// TIA Portal project "convergestation_Ronaldo" (V18)

(* hardware
DEVICE "S7-1200 station_1"  S7-1200 Station
   slot 0: "Rack_0"  S7-1200 Rack  Rack  V1.0
   slot 1: "Automacao_convergestation"  CPU 1214C DC/DC/DC  6ES7 214-1AG40-0XB0  V4.4
   slot 2: "DI 8/DQ 8x24VDC_1"  6ES7 223-1BH32-0XB0  V2.0
*)

// ===== PLC "Automacao_convergestation"  CPU 1214C DC/DC/DC =====

VAR_GLOBAL   // PLC tag table "Default tag table"
   "Emergência" AT %I0.0 : Bool;
   "Botão Start" AT %I0.1 : Bool;
   "Botão Stop" AT %I0.2 : Bool;
   "Botão Reset" AT %I0.3 : Bool;
   "Manual" AT %I0.4 : Bool;
   "Automático" AT %I0.5 : Bool;
   "Contador" AT %QD30 : DInt;
   "Clock_Byte" AT %MB0 : Byte;
   "Clock_10Hz" AT %M0.0 : Bool;
   "Clock_5Hz" AT %M0.1 : Bool;
   "Clock_2.5Hz" AT %M0.2 : Bool;
   "Clock_2Hz" AT %M0.3 : Bool;
   "Clock_1.25Hz" AT %M0.4 : Bool;
   "Clock_1Hz" AT %M0.5 : Bool;
   "Clock_0.625Hz" AT %M0.6 : Bool;
   "Clock_0.5Hz" AT %M0.7 : Bool;
   "Sen. Esteira 01" AT %I0.6 : Bool;
   "Sen. Esteira 02" AT %I0.7 : Bool;
   "Sen. Transf. 01" AT %I1.0 : Bool;
   "Sen. Transf. 02" AT %I1.1 : Bool;
   "Sen.  de Saída" AT %I1.2 : Bool;
   "Esteira 01" AT %Q0.0 : Bool;
   "Esteira 02" AT %Q0.1 : Bool;
   "Esteira de Saída" AT %Q0.2 : Bool;
   "Carregar 01" AT %Q0.3 : Bool;
   "Carregar 02" AT %Q0.4 : Bool;
   "Descarregar 01" AT %Q0.5 : Bool;
   "Descarregar 02" AT %Q0.6 : Bool;
   "Transf. 01 Direita" AT %Q0.7 : Bool;
   "Transf. 02 Direita" AT %Q1.0 : Bool;
   "Transf. 01 Esquerda" AT %Q1.1 : Bool;
   "Transf. 02 Esquerda" AT %Q1.2 : Bool;
   "Led Verde" AT %Q1.3 : Bool;
   "Led Amarelo" AT %Q1.4 : Bool;
   "Led Vermelho" AT %Q1.5 : Bool;
END_VAR

DATA_BLOCK "DB"   // DB1
{ S7_Optimized_Access := 'TRUE' }
VERSION : 0.1
   VAR
      Habilita : Bool;
      Ciclo_Automático : Bool;
      Auto : Bool;
      "M" : Array[0..6] of Bool;
      Ciclo_Manual : Bool;
      Block : Bool;
      "Rotina 01" : Bool;
      "Rotina 02" : Bool;
   END_VAR
BEGIN
END_DATA_BLOCK

// folder: System blocks/Program resources

DATA_BLOCK "Timer 0"   // DB2
{ S7_Optimized_Access := 'TRUE' }
AUTHOR : Simatic
FAMILY : IEC
NAME : IEC_TMR
VERSION : 1.0
// stored: InstanceOfName IEC_TIMER
"IEC_TIMER"
BEGIN
END_DATA_BLOCK

DATA_BLOCK "Timer 2"   // DB4
{ S7_Optimized_Access := 'TRUE' }
AUTHOR : Simatic
FAMILY : IEC
NAME : IEC_TMR
VERSION : 1.0
// stored: InstanceOfName IEC_TIMER
"IEC_TIMER"
BEGIN
END_DATA_BLOCK

DATA_BLOCK "Timer 3"   // DB5
{ S7_Optimized_Access := 'TRUE' }
AUTHOR : Simatic
FAMILY : IEC
NAME : IEC_TMR
VERSION : 1.0
// stored: InstanceOfName IEC_TIMER
"IEC_TIMER"
BEGIN
END_DATA_BLOCK

DATA_BLOCK "Timer 4"   // DB6
{ S7_Optimized_Access := 'TRUE' }
AUTHOR : Simatic
FAMILY : IEC
NAME : IEC_TMR
VERSION : 1.0
// stored: InstanceOfName IEC_TIMER
"IEC_TIMER"
BEGIN
END_DATA_BLOCK

DATA_BLOCK "Counter 0"   // DB8
{ S7_Optimized_Access := 'TRUE' }
AUTHOR : Simatic
FAMILY : IEC
NAME : CNTR
VERSION : 1.0
// stored: InstanceOfName IEC_COUNTER
"IEC_COUNTER"
BEGIN
END_DATA_BLOCK

// folder: (top level)

FUNCTION "PRINCIPAL" : Void   // FC1, LAD
{ S7_Optimized_Access := 'TRUE' }
VERSION : 0.1
   VAR_TEMP   // added for the SCL form of the ladder/FBD networks
      _w1 : Bool;
      _w2 : Bool;
      _w3 : Bool;
   END_VAR
BEGIN

REGION Network 1: Lógica de Emergência
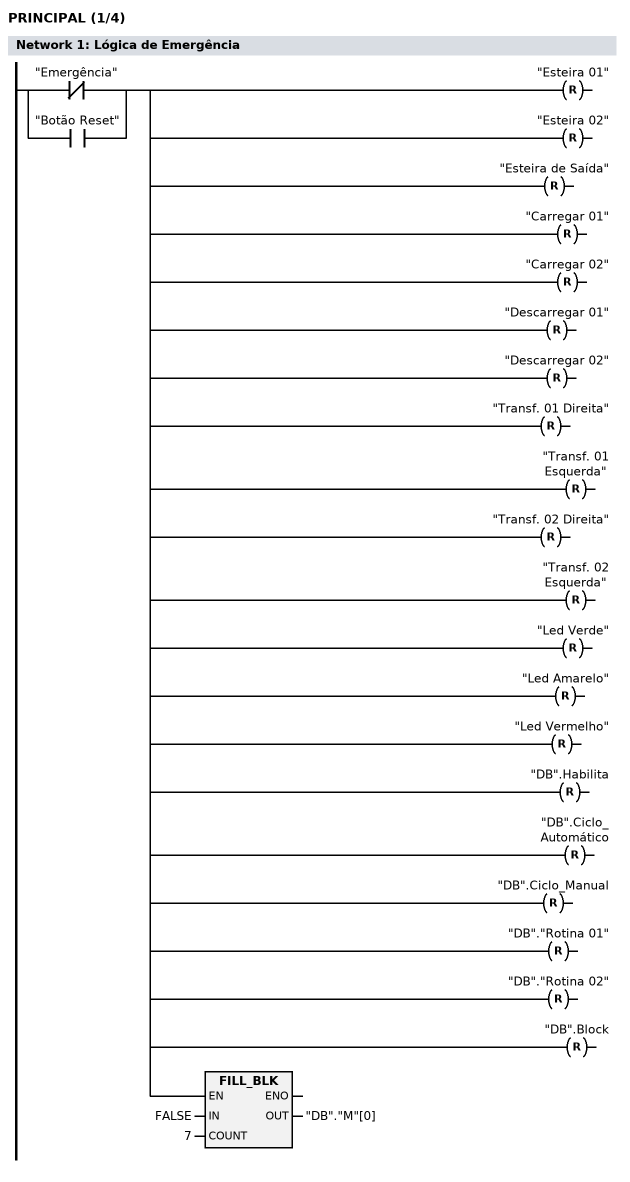
   RUNG wire#powerrail
      I_Contact( "Emergência" )
      wire#w1
      R_Coil( "Esteira 01" )
   END_RUNG
   RUNG wire#powerrail
      Contact( "Botão Reset" )
   END_RUNG wire#w1
   RUNG wire#w1
      R_Coil( "Esteira 02" )
   END_RUNG
   RUNG wire#w1
      R_Coil( "Esteira de Saída" )
   END_RUNG
   RUNG wire#w1
      R_Coil( "Carregar 01" )
   END_RUNG
   RUNG wire#w1
      R_Coil( "Carregar 02" )
   END_RUNG
   RUNG wire#w1
      R_Coil( "Descarregar 01" )
   END_RUNG
   RUNG wire#w1
      R_Coil( "Descarregar 02" )
   END_RUNG
   RUNG wire#w1
      R_Coil( "Transf. 01 Direita" )
   END_RUNG
   RUNG wire#w1
      R_Coil( "Transf. 01 Esquerda" )
   END_RUNG
   RUNG wire#w1
      R_Coil( "Transf. 02 Direita" )
   END_RUNG
   RUNG wire#w1
      R_Coil( "Transf. 02 Esquerda" )
   END_RUNG
   RUNG wire#w1
      R_Coil( "Led Verde" )
   END_RUNG
   RUNG wire#w1
      R_Coil( "Led Amarelo" )
   END_RUNG
   RUNG wire#w1
      R_Coil( "Led Vermelho" )
   END_RUNG
   RUNG wire#w1
      R_Coil( "DB".Habilita )
   END_RUNG
   RUNG wire#w1
      R_Coil( "DB".Ciclo_Automático )
   END_RUNG
   RUNG wire#w1
      R_Coil( "DB".Ciclo_Manual )
   END_RUNG
   RUNG wire#w1
      R_Coil( "DB"."Rotina 01" )
   END_RUNG
   RUNG wire#w1
      R_Coil( "DB"."Rotina 02" )
   END_RUNG
   RUNG wire#w1
      R_Coil( "DB".Block )
   END_RUNG
   RUNG wire#w1
      FillBlockI(in := FALSE, count := 7, out => "DB"."M"[0])
   END_RUNG
   // the same network as SCL:
   IF NOT "Emergência" OR "Botão Reset" THEN
       "Esteira 01" := FALSE;
       "Esteira 02" := FALSE;
       "Esteira de Saída" := FALSE;
       "Carregar 01" := FALSE;
       "Carregar 02" := FALSE;
       "Descarregar 01" := FALSE;
       "Descarregar 02" := FALSE;
       "Transf. 01 Direita" := FALSE;
       "Transf. 01 Esquerda" := FALSE;
       "Transf. 02 Direita" := FALSE;
       "Transf. 02 Esquerda" := FALSE;
       "Led Verde" := FALSE;
       "Led Amarelo" := FALSE;
       "Led Vermelho" := FALSE;
       "DB".Habilita := FALSE;
       "DB".Ciclo_Automático := FALSE;
       "DB".Ciclo_Manual := FALSE;
       "DB"."Rotina 01" := FALSE;
       "DB"."Rotina 02" := FALSE;
       "DB".Block := FALSE;
       FILL_BLK(IN := FALSE, COUNT := 7, OUT => "DB"."M"[0]);
   END_IF;
END_REGION

REGION Network 2: Lógica de Acionamentos Manuais
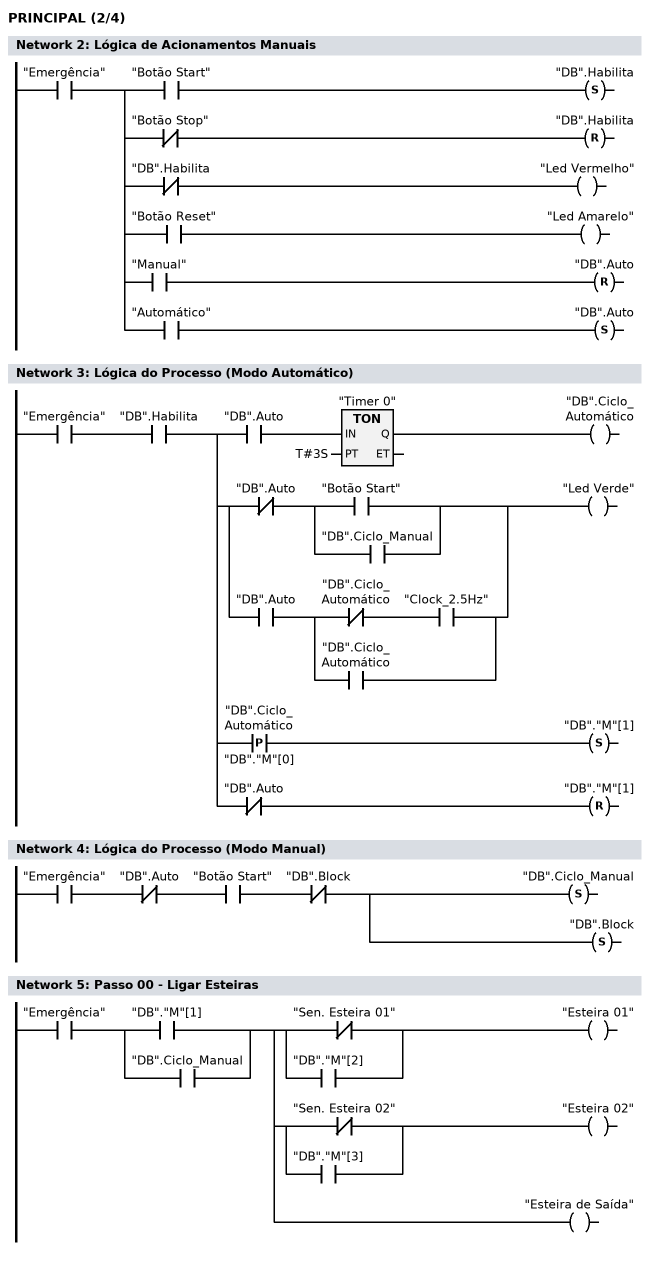
   RUNG wire#powerrail
      Contact( "Emergência" )
      wire#w1
      Contact( "Botão Start" )
      S_Coil( "DB".Habilita )
   END_RUNG
   RUNG wire#w1
      I_Contact( "Botão Stop" )
      R_Coil( "DB".Habilita )
   END_RUNG
   RUNG wire#w1
      I_Contact( "DB".Habilita )
      Coil( "Led Vermelho" )
   END_RUNG
   RUNG wire#w1
      Contact( "Botão Reset" )
      Coil( "Led Amarelo" )
   END_RUNG
   RUNG wire#w1
      Contact( "Manual" )
      R_Coil( "DB".Auto )
   END_RUNG
   RUNG wire#w1
      Contact( "Automático" )
      S_Coil( "DB".Auto )
   END_RUNG
   // the same network as SCL:
   IF "Emergência" AND "Botão Start" THEN "DB".Habilita := TRUE; END_IF;
   IF "Emergência" AND NOT "Botão Stop" THEN "DB".Habilita := FALSE; END_IF;
   "Led Vermelho" := "Emergência" AND NOT "DB".Habilita;
   "Led Amarelo" := "Emergência" AND "Botão Reset";
   IF "Emergência" AND "Manual" THEN "DB".Auto := FALSE; END_IF;
   IF "Emergência" AND "Automático" THEN "DB".Auto := TRUE; END_IF;
END_REGION

REGION Network 3: Lógica do Processo (Modo Automático)
   #_w1 := "Emergência" AND "DB".Habilita;
   "Timer 0".TON(IN := #_w1 AND "DB".Auto, PT := T#3S);
   "DB".Ciclo_Automático := "Timer 0".Q;
   "Led Verde" := #_w1 AND ((NOT "DB".Auto AND ("Botão Start" OR "DB".Ciclo_Manual)) OR ("DB".Auto AND ((NOT "DB".Ciclo_Automático AND "Clock_2.5Hz") OR "DB".Ciclo_Automático)));
   #_w2 := #_w1 AND "DB".Ciclo_Automático AND NOT "DB"."M"[0];   // rising edge of "DB".Ciclo_Automático
   "DB"."M"[0] := "DB".Ciclo_Automático;
   IF #_w2 THEN "DB"."M"[1] := TRUE; END_IF;
   IF #_w1 AND NOT "DB".Auto THEN "DB"."M"[1] := FALSE; END_IF;
END_REGION

REGION Network 4: Lógica do Processo (Modo Manual)
   RUNG wire#powerrail
      Contact( "Emergência" )
      I_Contact( "DB".Auto )
      Contact( "Botão Start" )
      I_Contact( "DB".Block )
      wire#w1
      S_Coil( "DB".Ciclo_Manual )
   END_RUNG
   RUNG wire#w1
      S_Coil( "DB".Block )
   END_RUNG
   // the same network as SCL:
   IF "Emergência" AND NOT "DB".Auto AND "Botão Start" AND NOT "DB".Block THEN
       "DB".Ciclo_Manual := TRUE;
       "DB".Block := TRUE;
   END_IF;
END_REGION

REGION Network 5: Passo 00 - Ligar Esteiras
   RUNG wire#powerrail
      Contact( "Emergência" )
      wire#w1
      Contact( "DB"."M"[1] )
      wire#w2
      I_Contact( "Sen. Esteira 01" )
      wire#w3
      Coil( "Esteira 01" )
   END_RUNG
   RUNG wire#w1
      Contact( "DB".Ciclo_Manual )
   END_RUNG wire#w2
   RUNG wire#w2
      Contact( "DB"."M"[2] )
   END_RUNG wire#w3
   RUNG wire#w2
      I_Contact( "Sen. Esteira 02" )
      wire#w4
      Coil( "Esteira 02" )
   END_RUNG
   RUNG wire#w2
      Contact( "DB"."M"[3] )
   END_RUNG wire#w4
   RUNG wire#w2
      Coil( "Esteira de Saída" )
   END_RUNG
   // the same network as SCL:
   #_w1 := "Emergência" AND ("DB"."M"[1] OR "DB".Ciclo_Manual);
   "Esteira 01" := #_w1 AND (NOT "Sen. Esteira 01" OR "DB"."M"[2]);
   "Esteira 02" := #_w1 AND (NOT "Sen. Esteira 02" OR "DB"."M"[3]);
   "Esteira de Saída" := #_w1;
END_REGION

REGION Network 6: Passo 01 - Identificar objeto e realizar para das Esteiras Correspondentes
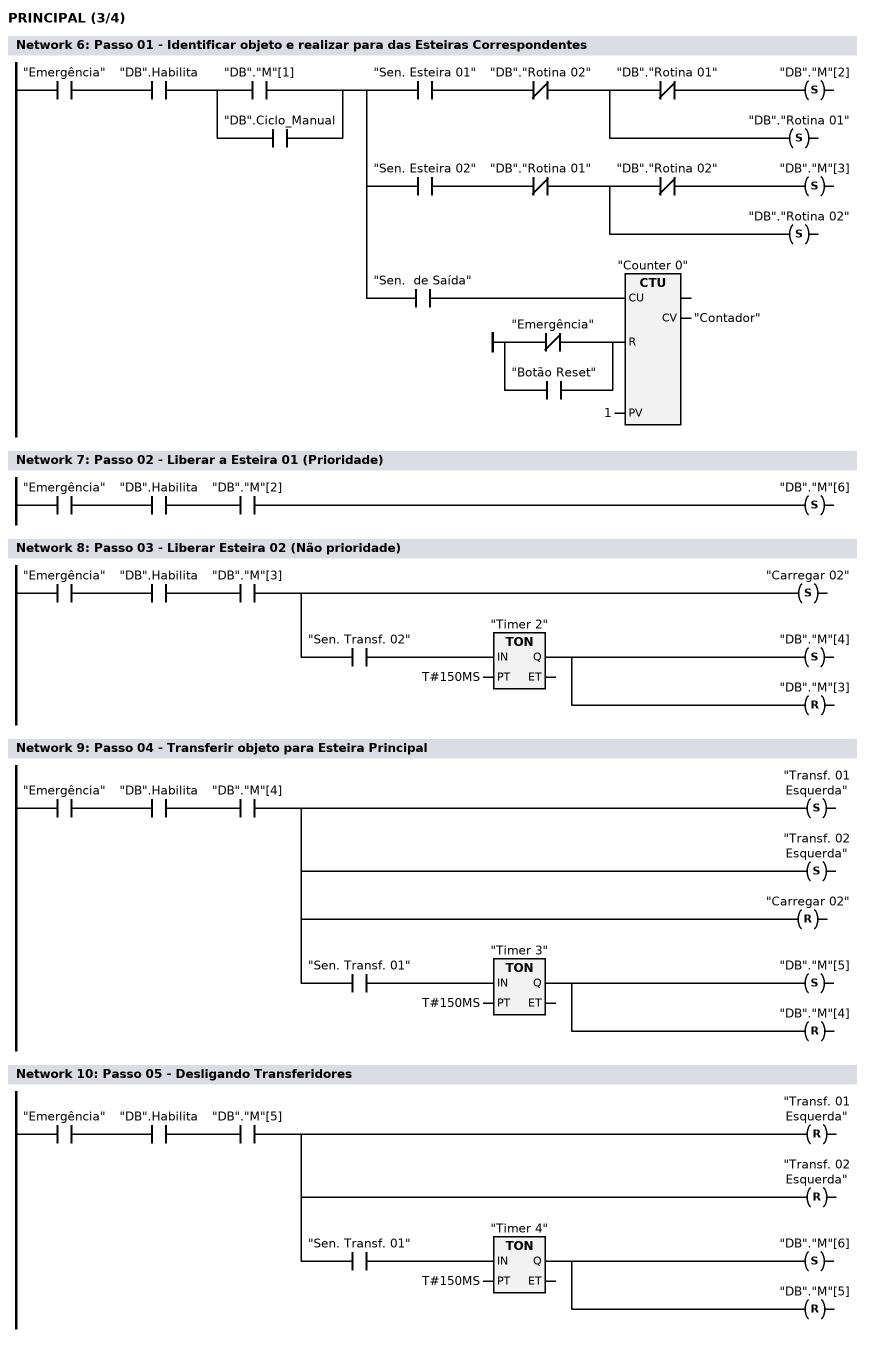
   #_w1 := "Emergência" AND "DB".Habilita AND ("DB"."M"[1] OR "DB".Ciclo_Manual);
   #_w2 := #_w1 AND "Sen. Esteira 01" AND NOT "DB"."Rotina 02";
   IF #_w2 AND NOT "DB"."Rotina 01" THEN "DB"."M"[2] := TRUE; END_IF;
   IF #_w2 THEN "DB"."Rotina 01" := TRUE; END_IF;
   #_w3 := #_w1 AND "Sen. Esteira 02" AND NOT "DB"."Rotina 01";
   IF #_w3 AND NOT "DB"."Rotina 02" THEN "DB"."M"[3] := TRUE; END_IF;
   IF #_w3 THEN "DB"."Rotina 02" := TRUE; END_IF;
   "Counter 0".CTU(CU := #_w1 AND "Sen.  de Saída",
                   R := NOT "Emergência" OR "Botão Reset",
                   PV := 1,
                   CV => "Contador");
END_REGION

REGION Network 7: Passo 02 - Liberar a Esteira 01 (Prioridade)
   RUNG wire#powerrail
      Contact( "Emergência" )
      Contact( "DB".Habilita )
      Contact( "DB"."M"[2] )
      S_Coil( "DB"."M"[6] )
   END_RUNG
   // the same network as SCL:
   IF "Emergência" AND "DB".Habilita AND "DB"."M"[2] THEN "DB"."M"[6] := TRUE; END_IF;
END_REGION

REGION Network 8: Passo 03 - Liberar Esteira 02 (Não prioridade)
   #_w1 := "Emergência" AND "DB".Habilita AND "DB"."M"[3];
   IF #_w1 THEN "Carregar 02" := TRUE; END_IF;
   "Timer 2".TON(IN := #_w1 AND "Sen. Transf. 02", PT := T#150MS);
   IF "Timer 2".Q THEN
       "DB"."M"[4] := TRUE;
       "DB"."M"[3] := FALSE;
   END_IF;
END_REGION

REGION Network 9: Passo 04 - Transferir objeto para Esteira Principal
   #_w1 := "Emergência" AND "DB".Habilita AND "DB"."M"[4];
   IF #_w1 THEN
       "Transf. 01 Esquerda" := TRUE;
       "Transf. 02 Esquerda" := TRUE;
       "Carregar 02" := FALSE;
   END_IF;
   "Timer 3".TON(IN := #_w1 AND "Sen. Transf. 01", PT := T#150MS);
   IF "Timer 3".Q THEN
       "DB"."M"[5] := TRUE;
       "DB"."M"[4] := FALSE;
   END_IF;
END_REGION

REGION Network 10: Passo 05 - Desligando Transferidores
   #_w1 := "Emergência" AND "DB".Habilita AND "DB"."M"[5];
   IF #_w1 THEN
       "Transf. 01 Esquerda" := FALSE;
       "Transf. 02 Esquerda" := FALSE;
   END_IF;
   "Timer 4".TON(IN := #_w1 AND "Sen. Transf. 01", PT := T#150MS);
   IF "Timer 4".Q THEN
       "DB"."M"[6] := TRUE;
       "DB"."M"[5] := FALSE;
   END_IF;
END_REGION

REGION Network 11: Passo 06 - Movendo o objeto Transferido para Esteira de Saída
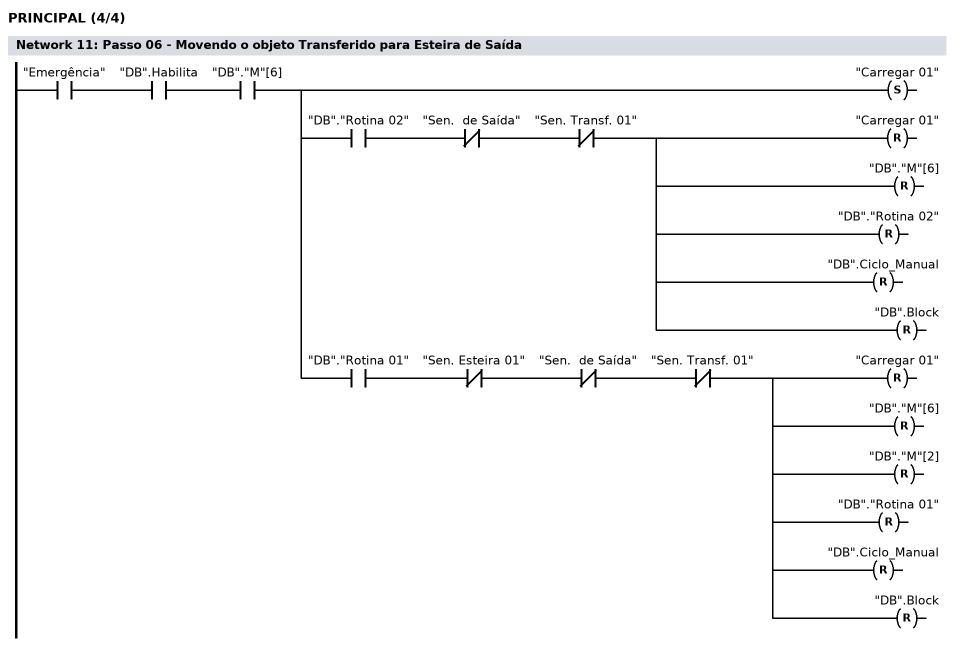
   RUNG wire#powerrail
      Contact( "Emergência" )
      Contact( "DB".Habilita )
      Contact( "DB"."M"[6] )
      wire#w1
      S_Coil( "Carregar 01" )
   END_RUNG
   RUNG wire#w1
      Contact( "DB"."Rotina 02" )
      I_Contact( "Sen.  de Saída" )
      I_Contact( "Sen. Transf. 01" )
      wire#w2
      R_Coil( "Carregar 01" )
   END_RUNG
   RUNG wire#w2
      R_Coil( "DB"."M"[6] )
   END_RUNG
   RUNG wire#w2
      R_Coil( "DB"."Rotina 02" )
   END_RUNG
   RUNG wire#w2
      R_Coil( "DB".Ciclo_Manual )
   END_RUNG
   RUNG wire#w2
      R_Coil( "DB".Block )
   END_RUNG
   RUNG wire#w1
      Contact( "DB"."Rotina 01" )
      I_Contact( "Sen. Esteira 01" )
      I_Contact( "Sen.  de Saída" )
      I_Contact( "Sen. Transf. 01" )
      wire#w3
      R_Coil( "Carregar 01" )
   END_RUNG
   RUNG wire#w3
      R_Coil( "DB"."M"[6] )
   END_RUNG
   RUNG wire#w3
      R_Coil( "DB"."M"[2] )
   END_RUNG
   RUNG wire#w3
      R_Coil( "DB"."Rotina 01" )
   END_RUNG
   RUNG wire#w3
      R_Coil( "DB".Ciclo_Manual )
   END_RUNG
   RUNG wire#w3
      R_Coil( "DB".Block )
   END_RUNG
   // the same network as SCL:
   #_w1 := "Emergência" AND "DB".Habilita AND "DB"."M"[6];
   IF #_w1 THEN "Carregar 01" := TRUE; END_IF;
   IF #_w1 AND "DB"."Rotina 02" AND NOT "Sen.  de Saída" AND NOT "Sen. Transf. 01" THEN
       "Carregar 01" := FALSE;
       "DB"."M"[6] := FALSE;
   END_IF;
   #_w2 := #_w1 AND "DB"."Rotina 02" AND NOT "Sen.  de Saída" AND NOT "Sen. Transf. 01";
   IF #_w2 THEN
       "DB"."Rotina 02" := FALSE;
       "DB".Ciclo_Manual := FALSE;
       "DB".Block := FALSE;
   END_IF;
   IF #_w1 AND "DB"."Rotina 01" AND NOT "Sen. Esteira 01" AND NOT "Sen.  de Saída" AND NOT "Sen. Transf. 01" THEN
       "Carregar 01" := FALSE;
       "DB"."M"[6] := FALSE;
       "DB"."M"[2] := FALSE;
   END_IF;
   #_w3 := #_w1 AND "DB"."Rotina 01" AND NOT "Sen. Esteira 01" AND NOT "Sen.  de Saída" AND NOT "Sen. Transf. 01";
   IF #_w3 THEN
       "DB"."Rotina 01" := FALSE;
       "DB".Ciclo_Manual := FALSE;
       "DB".Block := FALSE;
   END_IF;
END_REGION
END_FUNCTION

FUNCTION "MHJ-PLC-Lab-Function-S71200" : Void   // FC9000, SCL
{ S7_Optimized_Access := 'TRUE' }
VERSION : 0.1
   VAR_TEMP
      rdTimeReturn : Int;
      outputTime : DTL;
      SyncVal : Byte;
      forVal : Int;
      forVal_2 : Int;
      Value : Byte;
   END_VAR
   VAR CONSTANT
      CompVal : Byte := 16#34;
      Value_01 : Byte := 16#11;
      Value_01_DW : DWord := 16#A165_D992;
      Value_02_DW : DWord := 16#58BE_4401;
   END_VAR
BEGIN

   #Value:=PEEK(area := 16#82,
        dbNumber := 0,
        byteOffset := 511);
   #Value := #Value + 1;

   POKE(area := 16#82,
        dbNumber := 0,
        byteOffset := 511,
        value := #Value);

   POKE(area:=16#81,
        dbNumber:=0,
        byteOffset:=1016,
        value:=#Value_01_DW);
   POKE(area := 16#81,
        dbNumber := 0,
        byteOffset := 1020,
        value := #Value_02_DW);

   POKE(area := 16#81,
        dbNumber := 0,
        byteOffset := 511,
        value := B#16#00);

   FOR #forVal := 0 TO 120 DO
       FOR #forVal_2:=0 TO 10 DO
           #rdTimeReturn:=RD_SYS_T(#outputTime);
           #rdTimeReturn := WR_SYS_T(#outputTime);
           #rdTimeReturn := RD_SYS_T(#outputTime);
           #rdTimeReturn := WR_SYS_T(#outputTime);
       END_FOR;
       #SyncVal:= PEEK(area := 16#81,
                      dbNumber := 0,
                      byteOffset := 511);
       IF #SyncVal = #CompVal THEN
          GOTO M_1;
       END_IF;
   END_FOR;
   RETURN;

   M_1:
   POKE(area := 16#81,
        dbNumber := 0,
        byteOffset := 511,
        value := B#16#0);
END_FUNCTION

ORGANIZATION_BLOCK "Main"   // OB1, LAD, ProgramCycle
TITLE = "Main Program Sweep (Cycle)"
{ S7_Optimized_Access := 'TRUE' }
VERSION : 0.1
   VAR_INPUT
      Initial_Call : Bool;   // Initial call of this OB
      Remanence : Bool;   // =True, if remanent data are available
   END_VAR
BEGIN

REGION Network 1: Lógica de Comunicação
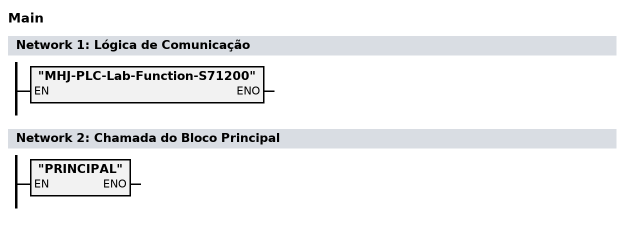
   RUNG wire#powerrail
      "MHJ-PLC-Lab-Function-S71200"()
   END_RUNG
   // the same network as SCL:
   "MHJ-PLC-Lab-Function-S71200"();
END_REGION

REGION Network 2: Chamada do Bloco Principal
   RUNG wire#powerrail
      "PRINCIPAL"()
   END_RUNG
   // the same network as SCL:
   "PRINCIPAL"();
END_REGION
END_ORGANIZATION_BLOCK